// TIA Portal project "w2_denGiaoThong1" (V14)

(* hardware
DEVICE "S7-1200 station_1"  S7-1200 Station
   slot 0: "Rack_0"  S7-1200 Rack  Rack  V1.0
   slot 1: "PLC_1"  CPU 1214C DC/DC/DC  6ES7 214-1AG40-0XB0  V4.2
DEVICE "HMI_1"  KTP700 Basic PN
   slot 0: "KTP700 Basic PN"  KTP700 Basic PN  6AV2 123-2GB03-0AX0  14.0.1.0
   slot 1: "HMI_RT_1"  KTP700 Basic PN  6AV2 123-2GB03-0AX0  14.0.1.0
   slot 5: "HMI_1.IE_CP_1"  PROFINET Interface  14.0.1.0
      slot 1: "PROFINET Interface_1"  PROFINET Interface
         slot 1: "Port_1"  Port
*)

// ===== PLC "PLC_1"  CPU 1214C DC/DC/DC =====

VAR_GLOBAL   // PLC tag table "Default tag table"
   "Daily" AT %M1.6 : Bool;
   "ngat" AT %M0.1 : Bool;
   "X1" AT %M0.2 : Bool;
   "V1" AT %M0.3 : Bool;
   "D1" AT %M0.4 : Bool;
   "sig1" AT %M0.0 : Bool;
   "Tag_1" AT %M0.7 : Bool;
   "ngat2" AT %M0.5 : Bool;
   "X2" AT %M0.6 : Bool;
   "D2" AT %M1.0 : Bool;
   "V2" AT %M1.1 : Bool;
   "Canh bao" AT %M1.7 : Bool;
   "sig2" AT %M1.2 : Bool;
   "UT" AT %M1.3 : Bool;
   "UT1" AT %M2.0 : Bool;
   "UT2" AT %M2.1 : Bool;
   "sig_ut1" AT %M1.4 : Bool;
   "sig_ut2" AT %M1.5 : Bool;
   "NX1" AT %M2.2 : Bool;
   "NV1" AT %M2.3 : Bool;
   "ND2" AT %M2.4 : Bool;
   "NX2" AT %M2.5 : Bool;
END_VAR

// folder: System blocks/Program resources

DATA_BLOCK "IEC_Timer_0_DB"   // DB1
{ S7_Optimized_Access := 'TRUE' }
AUTHOR : Simatic
FAMILY : IEC
NAME : IEC_TMR
VERSION : 1.0
// stored: InstanceOfName IEC_TIMER
"IEC_TIMER"
BEGIN
END_DATA_BLOCK

DATA_BLOCK "IEC_Timer0_DB"   // DB2
{ S7_Optimized_Access := 'TRUE' }
AUTHOR : Simatic
FAMILY : IEC
NAME : IEC_TMR
VERSION : 1.0
// stored: InstanceOfName IEC_TIMER
"IEC_TIMER"
BEGIN
END_DATA_BLOCK

DATA_BLOCK "IEC_Timer_0_DB_2"   // DB3
{ S7_Optimized_Access := 'TRUE' }
AUTHOR : Simatic
FAMILY : IEC
NAME : IEC_TMR
VERSION : 1.0
// stored: InstanceOfName IEC_TIMER
"IEC_TIMER"
BEGIN
END_DATA_BLOCK

DATA_BLOCK "IEC_Timer_DB_2"   // DB4
{ S7_Optimized_Access := 'TRUE' }
AUTHOR : Simatic
FAMILY : IEC
NAME : IEC_TMR
VERSION : 1.0
// stored: InstanceOfName IEC_TIMER
"IEC_TIMER"
BEGIN
END_DATA_BLOCK

DATA_BLOCK "IEC_Timer_0_DB_4"   // DB5
{ S7_Optimized_Access := 'TRUE' }
AUTHOR : Simatic
FAMILY : IEC
NAME : IEC_TMR
VERSION : 1.0
// stored: InstanceOfName IEC_TIMER
"IEC_TIMER"
BEGIN
END_DATA_BLOCK

DATA_BLOCK "IEC_Timer_0_DB_1"   // DB6
{ S7_Optimized_Access := 'TRUE' }
AUTHOR : Simatic
FAMILY : IEC
NAME : IEC_TMR
VERSION : 1.0
// stored: InstanceOfName IEC_TIMER
"IEC_TIMER"
BEGIN
END_DATA_BLOCK

DATA_BLOCK "IEC_Timer_0_DB_3"   // DB7
{ S7_Optimized_Access := 'TRUE' }
AUTHOR : Simatic
FAMILY : IEC
NAME : IEC_TMR
VERSION : 1.0
// stored: InstanceOfName IEC_TIMER
"IEC_TIMER"
BEGIN
END_DATA_BLOCK

DATA_BLOCK "IEC_Timer_0_DB_5"   // DB8
{ S7_Optimized_Access := 'TRUE' }
AUTHOR : Simatic
FAMILY : IEC
NAME : IEC_TMR
VERSION : 1.0
// stored: InstanceOfName IEC_TIMER
"IEC_TIMER"
BEGIN
END_DATA_BLOCK

// folder: (top level)

ORGANIZATION_BLOCK "Main"   // OB1, LAD, ProgramCycle
TITLE = "Main Program Sweep (Cycle)"
{ S7_Optimized_Access := 'TRUE' }
VERSION : 0.1
   VAR_INPUT
      Initial_Call : Bool;   // Initial call of this OB
      Remanence : Bool;   // =True, if remanent data are available
   END_VAR
   VAR_TEMP   // added for the SCL form of the ladder/FBD networks
      _w1 : Bool;
      _w2 : Bool;
      _w3 : Bool;
   END_VAR
BEGIN

REGION Network 1: Khi chua an nut uu tien
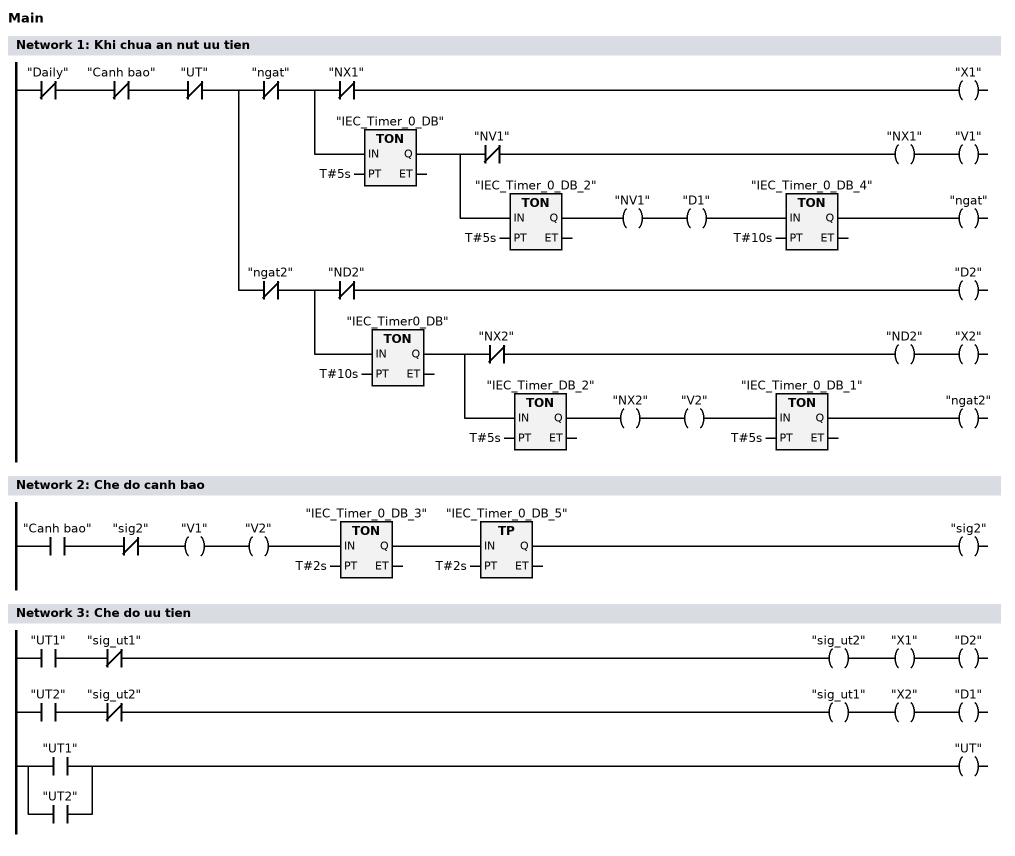
   #_w1 := NOT "Daily" AND NOT "Canh bao" AND NOT "UT";
   #_w2 := #_w1 AND NOT "ngat";
   "X1" := #_w2 AND NOT "NX1";
   "IEC_Timer_0_DB".TON(IN := #_w2, PT := T#5s);
   "NX1" := "IEC_Timer_0_DB".Q AND NOT "NV1";
   "V1" := "NX1";
   "IEC_Timer_0_DB_2".TON(IN := "IEC_Timer_0_DB".Q, PT := T#5s);
   "NV1" := "IEC_Timer_0_DB_2".Q;
   "D1" := "IEC_Timer_0_DB_2".Q;
   "IEC_Timer_0_DB_4".TON(IN := "IEC_Timer_0_DB_2".Q, PT := T#10s);
   "ngat" := "IEC_Timer_0_DB_4".Q;
   #_w3 := #_w1 AND NOT "ngat2";
   "D2" := #_w3 AND NOT "ND2";
   "IEC_Timer0_DB".TON(IN := #_w3, PT := T#10s);
   "ND2" := "IEC_Timer0_DB".Q AND NOT "NX2";
   "X2" := "ND2";
   "IEC_Timer_DB_2".TON(IN := "IEC_Timer0_DB".Q, PT := T#5s);
   "NX2" := "IEC_Timer_DB_2".Q;
   "V2" := "IEC_Timer_DB_2".Q;
   "IEC_Timer_0_DB_1".TON(IN := "IEC_Timer_DB_2".Q, PT := T#5s);
   "ngat2" := "IEC_Timer_0_DB_1".Q;
END_REGION

REGION Network 2: Che do canh bao
   "V1" := "Canh bao" AND NOT "sig2";
   "V2" := "V1";
   "IEC_Timer_0_DB_3".TON(IN := "V1", PT := T#2s);
   "IEC_Timer_0_DB_5".TP(IN := "IEC_Timer_0_DB_3".Q, PT := T#2s);
   "sig2" := "IEC_Timer_0_DB_5".Q;
END_REGION

REGION Network 3: Che do uu tien
   RUNG wire#powerrail
      Contact( "UT1" )
      I_Contact( "sig_ut1" )
      Coil( "sig_ut2" )
      Coil( "X1" )
      Coil( "D2" )
   END_RUNG
   RUNG wire#powerrail
      Contact( "UT2" )
      I_Contact( "sig_ut2" )
      Coil( "sig_ut1" )
      Coil( "X2" )
      Coil( "D1" )
   END_RUNG
   RUNG wire#powerrail
      Contact( "UT1" )
      wire#w1
      Coil( "UT" )
   END_RUNG
   RUNG wire#powerrail
      Contact( "UT2" )
   END_RUNG wire#w1
   // the same network as SCL:
   "sig_ut2" := "UT1" AND NOT "sig_ut1";
   "X1" := "sig_ut2";
   "D2" := "sig_ut2";
   "sig_ut1" := "UT2" AND NOT "sig_ut2";
   "X2" := "sig_ut1";
   "D1" := "sig_ut1";
   "UT" := "UT1" OR "UT2";
END_REGION
END_ORGANIZATION_BLOCK

(* ===== HMI "HMI_RT_1" =====
system functions are stored by id; their names below are inferred from use
connection "HMI_Connection_1": ETHERNET, SMART_S7_1200_OMS

HMI tags "Default tag table"
   "Tag_ScreenNumber" : UInt, internal
   "X1" : Bool = PLC X1 AT %M0.2, 1 s
   "V1" : Bool = PLC V1 AT %M0.3, 1 s
   "D1" : Bool = PLC D1 AT %M0.4, 1 s
   "X2" : Bool = PLC X2 AT %M0.6, 1 s
   "V2" : Bool = PLC V2 AT %M1.1, 1 s
   "D2" : Bool = PLC D2 AT %M1.0, 1 s
   "UT1" : Bool = PLC UT1 AT %M2.0, 1 s
   "UT2" : Bool = PLC UT2 AT %M2.1, 1 s
   "Daily" : Bool = PLC Daily AT %M1.6, 1 s
   "Canh bao" : Bool = PLC "Canh bao" AT %M1.7, 1 s

Template "Template_1" 800x480
   Button "Exit" at 714,429 size 71x50; TextOff 'Exit'; PictureOff "ExitRuntime_KTP700_Basic_PN_TR"; PictureOn "ExitRuntime_KTP700_Basic_PN_TR"
      on Release: StopRuntime(0)
   Button "Template_Button" at 614,429 size 71x50; TextOff 'Text'
   Button "Template_Button_1" at 514,429 size 71x50; TextOff 'Text'
   Button "Template_Button_2" at 414,429 size 71x50; TextOff 'Text'
   Button "Template_Button_3" at 314,429 size 71x50; TextOff 'Text'
   Button "Template_Button_4" at 214,429 size 71x50; TextOff 'Text'
   Button "Alarms" at 114,429 size 71x50; TextOff 'Alarms'; PictureOff "AlarmDisplay_KTP700_Basic_PN_TR"; PictureOn "AlarmDisplay_KTP700_Basic_PN_TR"
      on Release: function_ef3f5d25("Alarm window_Unacknowledged", -1)
   Button "Start screen" at 14,429 size 71x50; TextOff 'Start screen'; PictureOff "NavigateHome_KTP700_Basic_PN_TR"; PictureOn "NavigateHome_KTP700_Basic_PN_TR"
      on Release: ActivateScreen("Root screen", 0)
   SymbolicIOField "Symbolic_IO_Field_Screen" at 93,9 size 600x33; TextOff '0'; TextOn '1'; TextList "TextList_ScreenNames"
      ProcessValue <- "Tag_ScreenNumber"
      on Change: ActivateScreenByNumber("Tag_ScreenNumber", 0)
   DateTimeField "HmiScreenItemData" at 695,25 size 105x25
   DateTimeField "HmiScreenItemData_1" at 695,0 size 105x25
   GraphicView "Logo" at 0,0 size 91x51; Picture "Logo of HMI_1"

screen "Root screen" 800x480, template "Template_1"
   on GenerateScreen: SetTag("Tag_ScreenNumber", 1)
   Circle "Circle_1" at 401,38 size 23x23
      Appearance <- "X1"
   Circle "Circle_2" at 401,65 size 23x23
      Appearance <- "V1"
   Circle "Circle_3" at 401,95 size 23x23
      Appearance <- "D1"
   Circle "Circle_4" at 418,253 size 23x23
      Appearance <- "X2"
   Circle "Circle_5" at 418,280 size 23x23
      Appearance <- "V2"
   Circle "Circle_6" at 418,310 size 23x23
      Appearance <- "D2"
   IOField "I/O field_3" at 279,96 size 96x32; FormatPattern 1
      ProcessValue <- "UT1"
   IOField "I/O field_4" at 307,432 size 96x32; FormatPattern 1
      ProcessValue <- "UT2"
   Switch "Switch_1" at 27,134 size 64x32; CaptionText 'Switch'; TextOff 'OFF'; TextOn 'ON'
      on SwitchOn: SetBit("Daily")
      on SwitchOff: ResetBit("Daily")
   TextField "Text field_1" at 103,138 size 46x23; Text 'Daily'
   Switch "Switch_2" at 27,188 size 64x32; TextOn 'ON'; CaptionText 'Switch'; TextOff 'OFF'
      on SwitchOn: SetBit("Canh bao")
      on SwitchOff: ResetBit("Canh bao")
   TextField "Text field_2" at 105,192 size 51x23; Text 'warm'
   IOField "I/O field_1" at 20,96 size 96x32; FormatPattern 1
      ProcessValue <- "Daily"
   IOField "I/O field_2" at 20,244 size 96x32; FormatPattern 1
      ProcessValue <- "Canh bao"
   Switch "Switch_3" at 285,53 size 64x32; TextOn 'ON'; CaptionText 'Switch'; TextOff 'OFF'
      on SwitchOff: ResetBit("UT1")
      on SwitchOn: SetBit("UT1")
   Switch "Switch_4" at 313,384 size 64x32; TextOn 'ON'; CaptionText 'Switch'; TextOff 'OFF'
      on SwitchOff: ResetBit("UT2")
      on SwitchOn: SetBit("UT2")
*)